// Since FB_HasTaskInfo is an ABSTRACT class, the functionality needs to be implemented by extending the base class
FUNCTION_BLOCK INTERNAL FB_HasTaskInfo_ExtensionsForTests EXTENDS FB_HasTaskInfo
VAR_INPUT
END_VAR
VAR_OUTPUT
END_VAR
VAR
END_VAR

END_FUNCTION_BLOCK

(* stored: Version 1.1.0.1, ProductVersion 3.1.4024.13
   POU FB_HasTaskInfo_ExtensionsForTests: Id {039b3b48-b4ab-003b-21ce-ce2cfc334b7f}, SpecialFunc None *)
